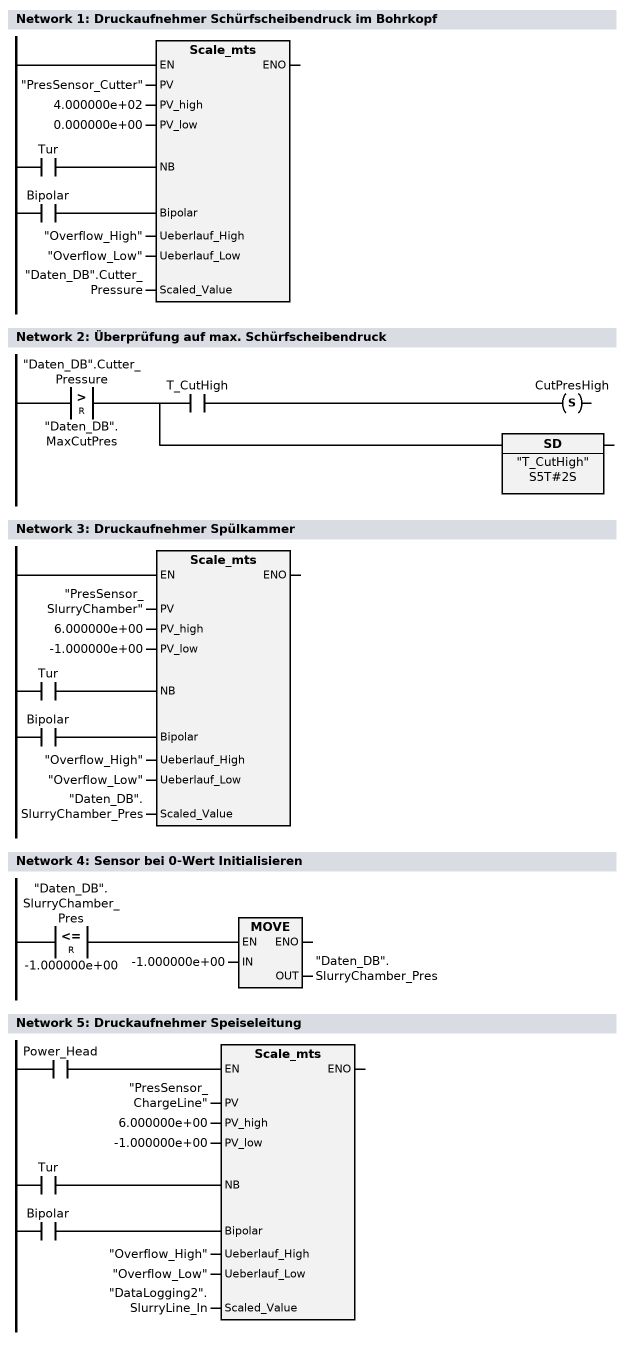
[picture p48: PresSensor_BK networks 1-5]
NETWORK
TITLE = Druckaufnehmer Schürfscheibendruck im Bohrkopf
      A     "Tur";
      =     L 0.0;
      BLD   103;
      A     "Bipolar";
      =     L 0.1;
      BLD   103;
      CALL  "Scale_mts" (
           PV                       := "PresSensor_Cutter",
           PV_high                  := 4.000000e+02,
           PV_low                   := 0.000000e+00,
           NB                       := L 0.0,
           Bipolar                  := L 0.1,
           Ueberlauf_High           := "Overflow_High",
           Ueberlauf_Low            := "Overflow_Low",
           Scaled_Value             := "Daten_DB".Cutter_Pressure);
      NOP   0;
NETWORK
TITLE = Überprüfung auf max. Schürfscheibendruck
      L     "Daten_DB".Cutter_Pressure;
      L     "Daten_DB".MaxCutPres;
      >R;
      =     L 0.0;
      A     L 0.0;
      A     "T_CutHigh";
      S     "CutPresHigh";
      A     L 0.0;
      BLD   102;
      L     S5T#2S;
      SD    "T_CutHigh";
NETWORK
TITLE = Druckaufnehmer Spülkammer
      A     "Tur";
      =     L 0.0;
      BLD   103;
      A     "Bipolar";
      =     L 0.1;
      BLD   103;
      CALL  "Scale_mts" (
           PV                       := "PresSensor_SlurryChamber",
           PV_high                  := 6.000000e+00,
           PV_low                   := -1.000000e+00,
           NB                       := L 0.0,
           Bipolar                  := L 0.1,
           Ueberlauf_High           := "Overflow_High",
           Ueberlauf_Low            := "Overflow_Low",
           Scaled_Value             := "Daten_DB".SlurryChamber_Pres);
      NOP   0;
NETWORK
TITLE = Sensor bei 0-Wert Initialisieren
      A(;
      L     "Daten_DB".SlurryChamber_Pres;
      L     -1.000000e+00;
      <=R;
      );
      JNB   _001;
      L     -1.000000e+00;
      T     "Daten_DB".SlurryChamber_Pres;
_001: NOP   0;
NETWORK
TITLE = Druckaufnehmer Speiseleitung
      A     "Tur";
      =     L 0.0;
      BLD   103;
      A     "Bipolar";
      =     L 0.1;
      BLD   103;
      A     "Power_Head";
      JNB   _002;
      CALL  "Scale_mts" (
           PV                       := "PresSensor_ChargeLine",
           PV_high                  := 6.000000e+00,
           PV_low                   := -1.000000e+00,
           NB                       := L 0.0,
           Bipolar                  := L 0.1,
           Ueberlauf_High           := "Overflow_High",
           Ueberlauf_Low            := "Overflow_Low",
           Scaled_Value             := "DataLogging2".SlurryLine_In);
_002: NOP   0;
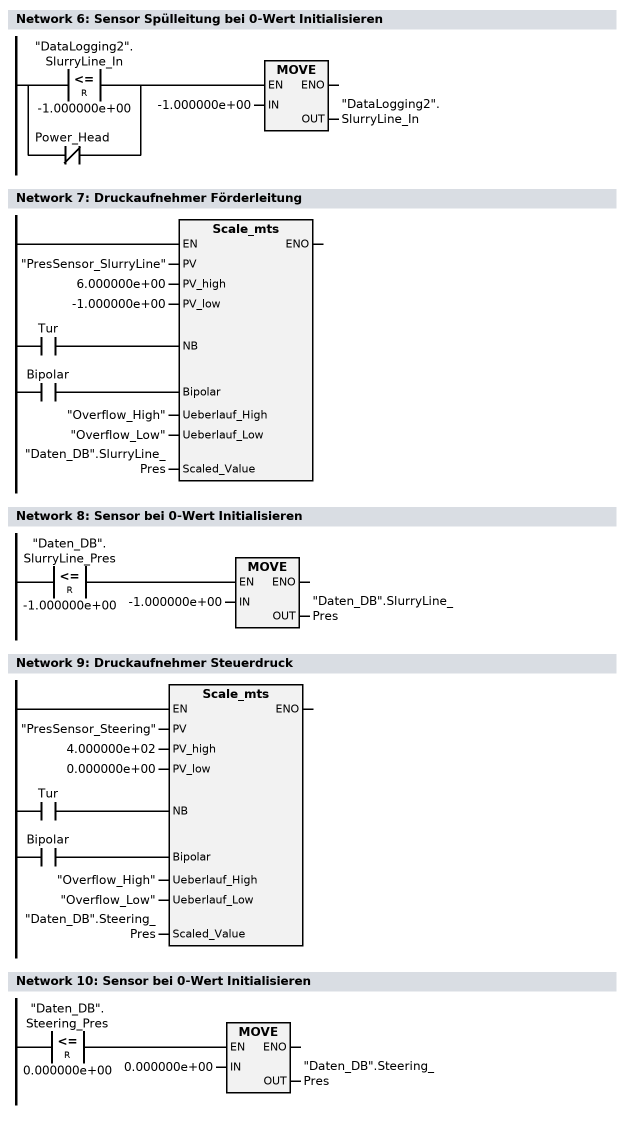
NETWORK
TITLE = Sensor Spülleitung bei 0-Wert Initialisieren
      A(;
      O(;
      L     "DataLogging2".SlurryLine_In;
      L     -1.000000e+00;
      <=R;
      );
      ON    "Power_Head";
      );
      JNB   _003;
      L     -1.000000e+00;
      T     "DataLogging2".SlurryLine_In;
_003: NOP   0;
NETWORK
TITLE = Druckaufnehmer Förderleitung
      A     "Tur";
      =     L 0.0;
      BLD   103;
      A     "Bipolar";
      =     L 0.1;
      BLD   103;
      CALL  "Scale_mts" (
           PV                       := "PresSensor_SlurryLine",
           PV_high                  := 6.000000e+00,
           PV_low                   := -1.000000e+00,
           NB                       := L 0.0,
           Bipolar                  := L 0.1,
           Ueberlauf_High           := "Overflow_High",
           Ueberlauf_Low            := "Overflow_Low",
           Scaled_Value             := "Daten_DB".SlurryLine_Pres);
      NOP   0;
NETWORK
TITLE = Sensor bei 0-Wert Initialisieren
      A(;
      L     "Daten_DB".SlurryLine_Pres;
      L     -1.000000e+00;
      <=R;
      );
      JNB   _004;
      L     -1.000000e+00;
      T     "Daten_DB".SlurryLine_Pres;
_004: NOP   0;
NETWORK
TITLE = Druckaufnehmer Steuerdruck
      A     "Tur";
      =     L 0.0;
      BLD   103;
      A     "Bipolar";
      =     L 0.1;
      BLD   103;
      CALL  "Scale_mts" (
           PV                       := "PresSensor_Steering",
           PV_high                  := 4.000000e+02,
           PV_low                   := 0.000000e+00,
           NB                       := L 0.0,
           Bipolar                  := L 0.1,
           Ueberlauf_High           := "Overflow_High",
           Ueberlauf_Low            := "Overflow_Low",
           Scaled_Value             := "Daten_DB".Steering_Pres);
      NOP   0;
NETWORK
TITLE = Sensor bei 0-Wert Initialisieren
      A(;
      L     "Daten_DB".Steering_Pres;
      L     0.000000e+00;
      <=R;
      );
      JNB   _005;
      L     0.000000e+00;
      T     "Daten_DB".Steering_Pres;
_005: NOP   0;
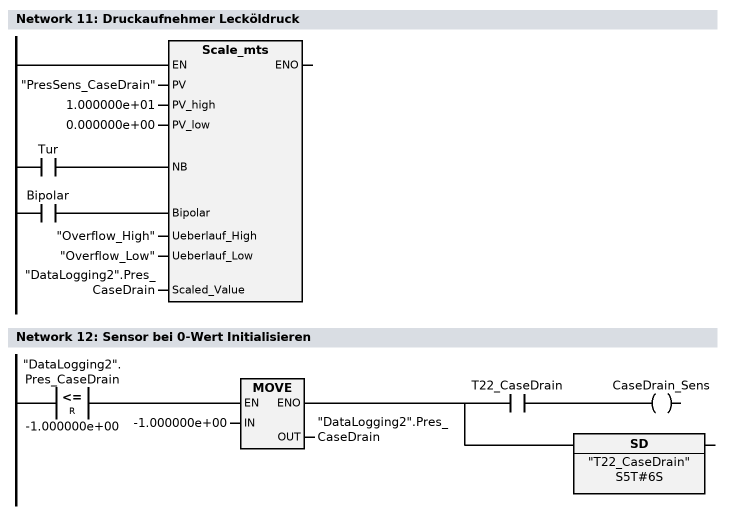
NETWORK
TITLE = Druckaufnehmer Lecköldruck
      A     "Tur";
      =     L 0.0;
      BLD   103;
      A     "Bipolar";
      =     L 0.1;
      BLD   103;
      CALL  "Scale_mts" (
           PV                       := "PresSens_CaseDrain",
           PV_high                  := 1.000000e+01,
           PV_low                   := 0.000000e+00,
           NB                       := L 0.0,
           Bipolar                  := L 0.1,
           Ueberlauf_High           := "Overflow_High",
           Ueberlauf_Low            := "Overflow_Low",
           Scaled_Value             := "DataLogging2".Pres_CaseDrain);
      NOP   0;
NETWORK
TITLE = Sensor bei 0-Wert Initialisieren
      A(;
      L     "DataLogging2".Pres_CaseDrain;
      L     -1.000000e+00;
      <=R;
      );
      JNB   _006;
      L     -1.000000e+00;
      T     "DataLogging2".Pres_CaseDrain;
      SET;
      SAVE;
      CLR;
_006: A     BR;
      =     L 0.0;
      A     L 0.0;
      A     "T22_CaseDrain";
      =     "CaseDrain_Sens";
      A     L 0.0;
      BLD   102;
      L     S5T#6S;
      SD    "T22_CaseDrain";
END_FUNCTION

FUNCTION "Steering cylinder 1" : VOID	// FC 40
TITLE = Funktionen für Steuerzylinder 1
AUTHOR : Simdon
FAMILY : Head
NAME : Cyl_1
VERSION : 0.1
VAR_TEMP
  ist : REAL ;	//Weg ohne Nullabgleich
  Fault : BOOL ;
  Stroke1 : DINT ;
  Stroke : REAL ;
END_VAR
BEGIN
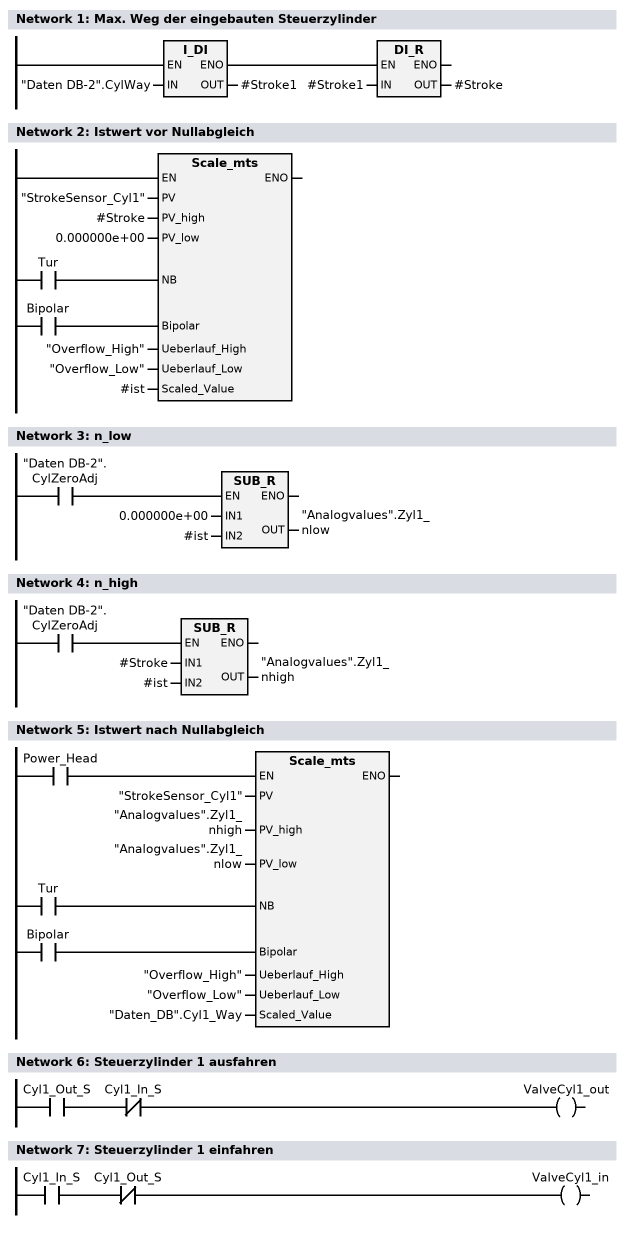
NETWORK
TITLE = Max. Weg der eingebauten Steuerzylinder
      A(;
      L     "Daten DB-2".CylWay;
      ITD;
      T     #Stroke1;
      SET;
      SAVE;
      CLR;
      A     BR;
      );
      JNB   _001;
      L     #Stroke1;
      DTR;
      T     #Stroke;
_001: NOP   0;
NETWORK
TITLE = Istwert vor Nullabgleich
//Istwert des Wegaufnehmers einlesen um die neue Unter- bzw. Obergrenze zur
//Bestimmung des Weges nach dem Nullabgleich. Die Wegaufnehmer liefern ein
//Signal von 4..20 mA.
      A     "Tur";
      =     L 14.0;
      BLD   103;
      A     "Bipolar";
      =     L 14.1;
      BLD   103;
      CALL  "Scale_mts" (
           PV                       := "StrokeSensor_Cyl1",
           PV_high                  := #Stroke,
           PV_low                   := 0.000000e+00,
           NB                       := L 14.0,
           Bipolar                  := L 14.1,
           Ueberlauf_High           := "Overflow_High",
           Ueberlauf_Low            := "Overflow_Low",
           Scaled_Value             := #ist);
      NOP   0;
NETWORK
TITLE = n_low
//Untergrenze der technischen Einheit nach durchgeführtem Nullabgleich.
      A     "Daten DB-2".CylZeroAdj;
      JNB   _002;
      L     0.000000e+00;
      L     #ist;
      -R;
      T     "Analogvalues".Zyl1_nlow;
_002: NOP   0;
NETWORK
TITLE = n_high
//Obergrenze der technischen Einheit nach durchgeführtem Nullabgleich.
      A     "Daten DB-2".CylZeroAdj;
      JNB   _003;
      L     #Stroke;
      L     #ist;
      -R;
      T     "Analogvalues".Zyl1_nhigh;
_003: NOP   0;
NETWORK
TITLE = Istwert nach Nullabgleich
//Istwert des Wegaufnehmers nach durchgeführtem Nullabgleich. Der Rückgabewert 
//liegt
//als Wert mit technischer Einheit (mm) vor.
      A     "Tur";
      =     L 14.0;
      BLD   103;
      A     "Bipolar";
      =     L 14.1;
      BLD   103;
      A     "Power_Head";
      JNB   _004;
      CALL  "Scale_mts" (
           PV                       := "StrokeSensor_Cyl1",
           PV_high                  := "Analogvalues".Zyl1_nhigh,
           PV_low                   := "Analogvalues".Zyl1_nlow,
           NB                       := L 14.0,
           Bipolar                  := L 14.1,
           Ueberlauf_High           := "Overflow_High",
           Ueberlauf_Low            := "Overflow_Low",
           Scaled_Value             := "Daten_DB".Cyl1_Way);
_004: NOP   0;
NETWORK
TITLE = Steuerzylinder 1 ausfahren
      A     "Cyl1_Out_S";
      AN    "Cyl1_In_S";
      =     "ValveCyl1_out";
NETWORK
TITLE = Steuerzylinder 1 einfahren
      A     "Cyl1_In_S";
      AN    "Cyl1_Out_S";
      =     "ValveCyl1_in";
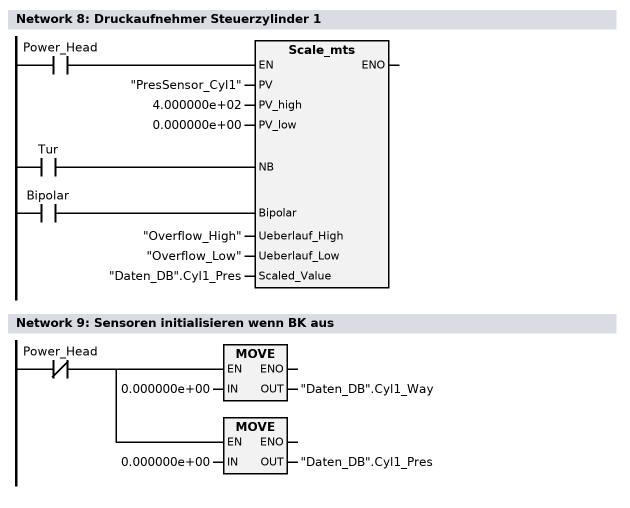
NETWORK
TITLE = Druckaufnehmer Steuerzylinder 1
      A     "Tur";
      =     L 14.0;
      BLD   103;
      A     "Bipolar";
      =     L 14.1;
      BLD   103;
      A     "Power_Head";
      JNB   _005;
      CALL  "Scale_mts" (
           PV                       := "PresSensor_Cyl1",
           PV_high                  := 4.000000e+02,
           PV_low                   := 0.000000e+00,
           NB                       := L 14.0,
           Bipolar                  := L 14.1,
           Ueberlauf_High           := "Overflow_High",
           Ueberlauf_Low            := "Overflow_Low",
           Scaled_Value             := "Daten_DB".Cyl1_Pres);
_005: NOP   0;
NETWORK
TITLE = Sensoren initialisieren wenn BK aus
      AN    "Power_Head";
      =     L 14.0;
      A     L 14.0;
      JNB   _006;
      L     0.000000e+00;
      T     "Daten_DB".Cyl1_Way;
_006: NOP   0;
      A     L 14.0;
      JNB   _007;
      L     0.000000e+00;
      T     "Daten_DB".Cyl1_Pres;
_007: NOP   0;
END_FUNCTION

FUNCTION "Steering cylinder 2" : VOID	// FC 41
TITLE = Funktionen für Steuerzylinder 2
AUTHOR : Simdon
FAMILY : Head
NAME : Cyl_2
VERSION : 0.1
VAR_TEMP
  ist : REAL ;	//Weg ohne Nullabgleich
  Fault : BOOL ;
  Stroke1 : DINT ;
  Stroke : REAL ;
END_VAR
BEGIN
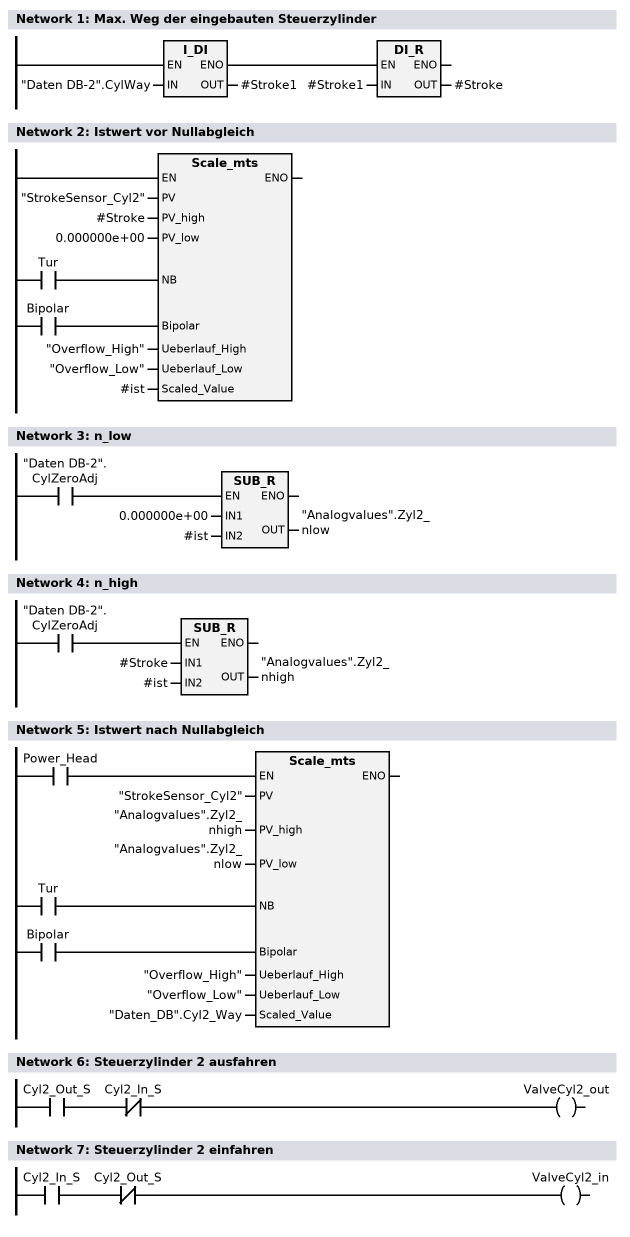
NETWORK
TITLE = Max. Weg der eingebauten Steuerzylinder
      A(;
      L     "Daten DB-2".CylWay;
      ITD;
      T     #Stroke1;
      SET;
      SAVE;
      CLR;
      A     BR;
      );
      JNB   _001;
      L     #Stroke1;
      DTR;
      T     #Stroke;
_001: NOP   0;
NETWORK
TITLE = Istwert vor Nullabgleich
//Istwert des Wegaufnehmers einlesen um die neue Unter- bzw. Obergrenze zur
//Bestimmung des Weges nach dem Nullabgleich. Die Wegaufnehmer liefern ein
//Signal von 4..20 mA.
      A     "Tur";
      =     L 14.0;
      BLD   103;
      A     "Bipolar";
      =     L 14.1;
      BLD   103;
      CALL  "Scale_mts" (
           PV                       := "StrokeSensor_Cyl2",
           PV_high                  := #Stroke,
           PV_low                   := 0.000000e+00,
           NB                       := L 14.0,
           Bipolar                  := L 14.1,
           Ueberlauf_High           := "Overflow_High",
           Ueberlauf_Low            := "Overflow_Low",
           Scaled_Value             := #ist);
      NOP   0;
NETWORK
TITLE = n_low
//Untergrenze der technischen Einheit nach durchgeführtem Nullabgleich.
      A     "Daten DB-2".CylZeroAdj;
      JNB   _002;
      L     0.000000e+00;
      L     #ist;
      -R;
      T     "Analogvalues".Zyl2_nlow;
_002: NOP   0;
NETWORK
TITLE = n_high
//Obergrenze der technischen Einheit nach durchgeführtem Nullabgleich.
      A     "Daten DB-2".CylZeroAdj;
      JNB   _003;
      L     #Stroke;
      L     #ist;
      -R;
      T     "Analogvalues".Zyl2_nhigh;
_003: NOP   0;
NETWORK
TITLE = Istwert nach Nullabgleich
//Istwert des Wegaufnehmers nach durchgeführtem Nullabgleich. Der Rückgabewert 
//liegt
//als Wert mit technischer Einheit (mm) vor.
      A     "Tur";
      =     L 14.0;
      BLD   103;
      A     "Bipolar";
      =     L 14.1;
      BLD   103;
      A     "Power_Head";
      JNB   _004;
      CALL  "Scale_mts" (
           PV                       := "StrokeSensor_Cyl2",
           PV_high                  := "Analogvalues".Zyl2_nhigh,
           PV_low                   := "Analogvalues".Zyl2_nlow,
           NB                       := L 14.0,
           Bipolar                  := L 14.1,
           Ueberlauf_High           := "Overflow_High",
           Ueberlauf_Low            := "Overflow_Low",
           Scaled_Value             := "Daten_DB".Cyl2_Way);
_004: NOP   0;
NETWORK
TITLE = Steuerzylinder 2 ausfahren
      A     "Cyl2_Out_S";
      AN    "Cyl2_In_S";
      =     "ValveCyl2_out";
NETWORK
TITLE = Steuerzylinder 2 einfahren
      A     "Cyl2_In_S";
      AN    "Cyl2_Out_S";
      =     "ValveCyl2_in";
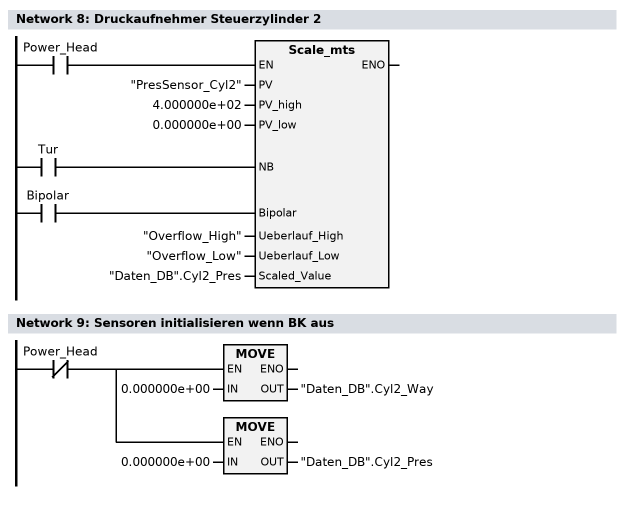
NETWORK
TITLE = Druckaufnehmer Steuerzylinder 2
      A     "Tur";
      =     L 14.0;
      BLD   103;
      A     "Bipolar";
      =     L 14.1;
      BLD   103;
      A     "Power_Head";
      JNB   _005;
      CALL  "Scale_mts" (
           PV                       := "PresSensor_Cyl2",
           PV_high                  := 4.000000e+02,
           PV_low                   := 0.000000e+00,
           NB                       := L 14.0,
           Bipolar                  := L 14.1,
           Ueberlauf_High           := "Overflow_High",
           Ueberlauf_Low            := "Overflow_Low",
           Scaled_Value             := "Daten_DB".Cyl2_Pres);
_005: NOP   0;
NETWORK
TITLE = Sensoren initialisieren wenn BK aus
      AN    "Power_Head";
      =     L 14.0;
      A     L 14.0;
      JNB   _006;
      L     0.000000e+00;
      T     "Daten_DB".Cyl2_Way;
_006: NOP   0;
      A     L 14.0;
      JNB   _007;
      L     0.000000e+00;
      T     "Daten_DB".Cyl2_Pres;
_007: NOP   0;
END_FUNCTION

FUNCTION "Steering cylinder 3" : VOID	// FC 42
TITLE = Funktionen für Steuerzylinder 3
AUTHOR : Simdon
FAMILY : Head
NAME : Cyl_3
VERSION : 0.1
VAR_TEMP
  ist : REAL ;	//Weg ohne Nullabgleich
  Fault : BOOL ;
  eins : INT ;
  Stroke1 : DINT ;
  Stroke : REAL ;
END_VAR
BEGIN
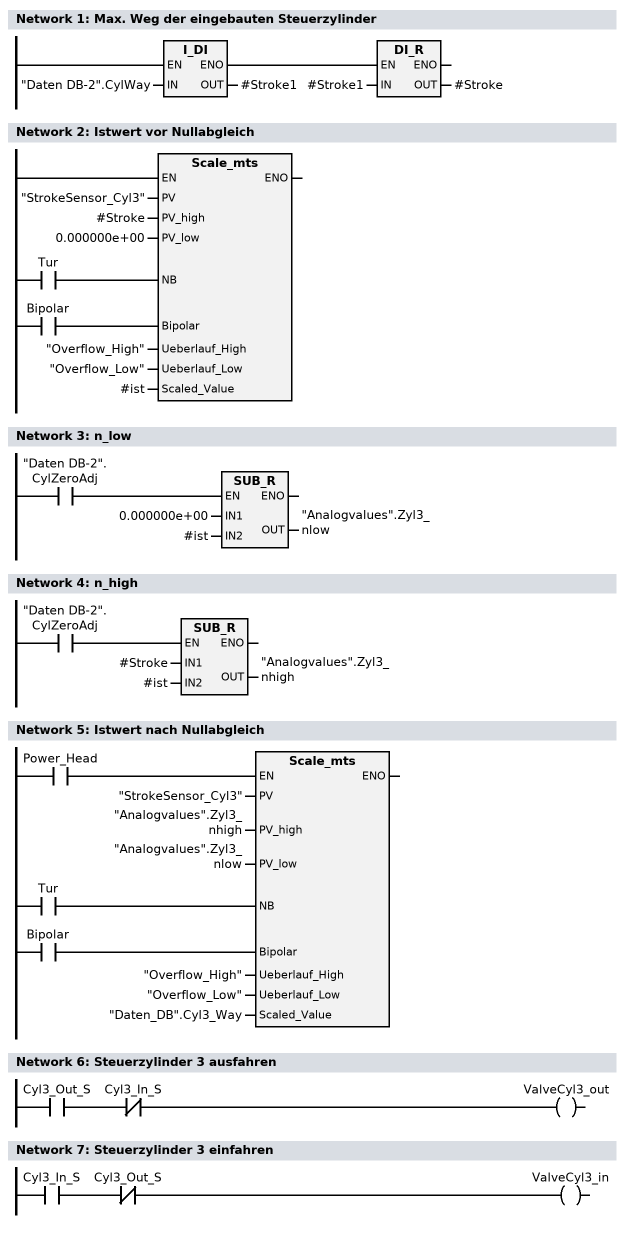
NETWORK
TITLE = Max. Weg der eingebauten Steuerzylinder
      A(;
      L     "Daten DB-2".CylWay;
      ITD;
      T     #Stroke1;
      SET;
      SAVE;
      CLR;
      A     BR;
      );
      JNB   _001;
      L     #Stroke1;
      DTR;
      T     #Stroke;
_001: NOP   0;
NETWORK
TITLE = Istwert vor Nullabgleich
//Istwert des Wegaufnehmers einlesen um die neue Unter- bzw. Obergrenze zur
//Bestimmung des Weges nach dem Nullabgleich. Die Wegaufnehmer liefern ein
//Signal von 4..20 mA.
      A     "Tur";
      =     L 16.0;
      BLD   103;
      A     "Bipolar";
      =     L 16.1;
      BLD   103;
      CALL  "Scale_mts" (
           PV                       := "StrokeSensor_Cyl3",
           PV_high                  := #Stroke,
           PV_low                   := 0.000000e+00,
           NB                       := L 16.0,
           Bipolar                  := L 16.1,
           Ueberlauf_High           := "Overflow_High",
           Ueberlauf_Low            := "Overflow_Low",
           Scaled_Value             := #ist);
      NOP   0;
NETWORK
TITLE = n_low
//Untergrenze der technischen Einheit nach durchgeführtem Nullabgleich.
      A     "Daten DB-2".CylZeroAdj;
      JNB   _002;
      L     0.000000e+00;
      L     #ist;
      -R;
      T     "Analogvalues".Zyl3_nlow;
_002: NOP   0;
NETWORK
TITLE = n_high
//Obergrenze der technischen Einheit nach durchgeführtem Nullabgleich.
      A     "Daten DB-2".CylZeroAdj;
      JNB   _003;
      L     #Stroke;
      L     #ist;
      -R;
      T     "Analogvalues".Zyl3_nhigh;
_003: NOP   0;
NETWORK
TITLE = Istwert nach Nullabgleich
//Istwert des Wegaufnehmers nach durchgeführtem Nullabgleich. Der Rückgabewert 
//liegt
//als Wert mit technischer Einheit (mm) vor.
      A     "Tur";
      =     L 16.0;
      BLD   103;
      A     "Bipolar";
      =     L 16.1;
      BLD   103;
      A     "Power_Head";
      JNB   _004;
      CALL  "Scale_mts" (
           PV                       := "StrokeSensor_Cyl3",
           PV_high                  := "Analogvalues".Zyl3_nhigh,
           PV_low                   := "Analogvalues".Zyl3_nlow,
           NB                       := L 16.0,
           Bipolar                  := L 16.1,
           Ueberlauf_High           := "Overflow_High",
           Ueberlauf_Low            := "Overflow_Low",
           Scaled_Value             := "Daten_DB".Cyl3_Way);
_004: NOP   0;
NETWORK
TITLE = Steuerzylinder 3 ausfahren
      A     "Cyl3_Out_S";
      AN    "Cyl3_In_S";
      =     "ValveCyl3_out";
NETWORK
TITLE = Steuerzylinder 3 einfahren
      A     "Cyl3_In_S";
      AN    "Cyl3_Out_S";
      =     "ValveCyl3_in";
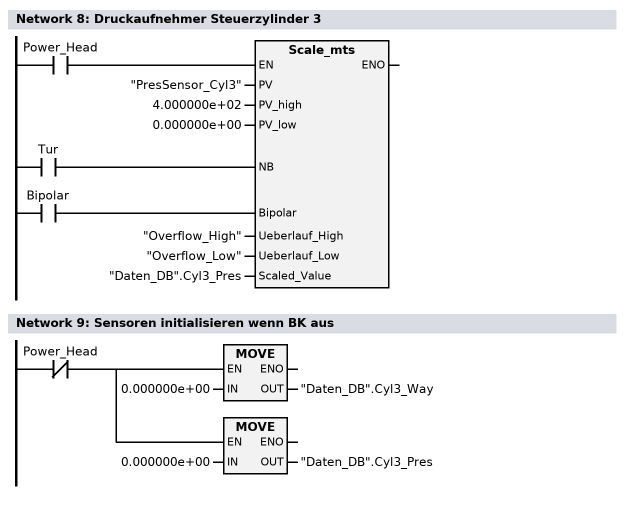
NETWORK
TITLE = Druckaufnehmer Steuerzylinder 3
      A     "Tur";
      =     L 16.0;
      BLD   103;
      A     "Bipolar";
      =     L 16.1;
      BLD   103;
      A     "Power_Head";
      JNB   _005;
      CALL  "Scale_mts" (
           PV                       := "PresSensor_Cyl3",
           PV_high                  := 4.000000e+02,
           PV_low                   := 0.000000e+00,
           NB                       := L 16.0,
           Bipolar                  := L 16.1,
           Ueberlauf_High           := "Overflow_High",
           Ueberlauf_Low            := "Overflow_Low",
           Scaled_Value             := "Daten_DB".Cyl3_Pres);
_005: NOP   0;
NETWORK
TITLE = Sensoren initialisieren wenn BK aus
      AN    "Power_Head";
      =     L 16.0;
      A     L 16.0;
      JNB   _006;
      L     0.000000e+00;
      T     "Daten_DB".Cyl3_Way;
_006: NOP   0;
      A     L 16.0;
      JNB   _007;
      L     0.000000e+00;
      T     "Daten_DB".Cyl3_Pres;
_007: NOP   0;
END_FUNCTION

FUNCTION "Wing" : VOID	// FC 43
TITLE = Funktionen für Flossenzylinder
AUTHOR : Simdon
FAMILY : Head
NAME : Wing
VERSION : 0.1
VAR_TEMP
  ist : REAL ;	//Weg ohne Nullabgleich
  Fault : BOOL ;
END_VAR
BEGIN
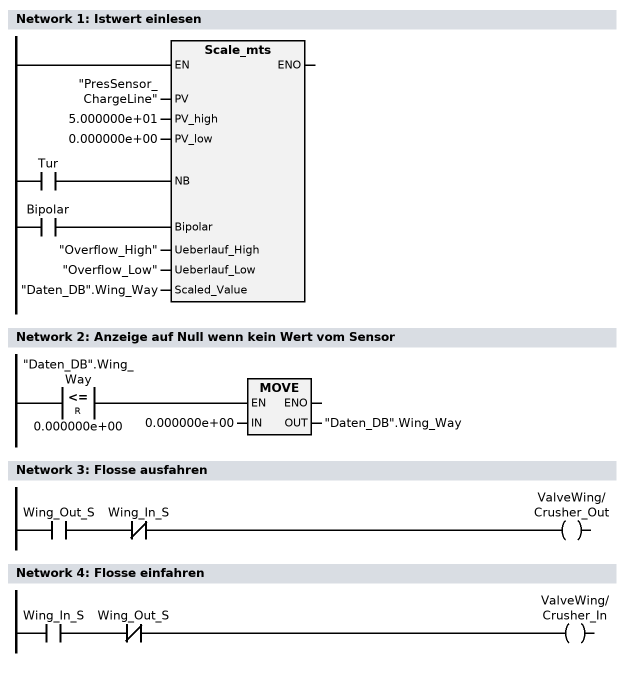
NETWORK
TITLE = Istwert einlesen
//Istwert des Wegaufnehmers nach durchgeführtem Nullabgleich. Der Rückgabewert 
//liegt
//als Wert mit technischer Einheit (mm) vor.
      A     "Tur";
      =     L 5.0;
      BLD   103;
      A     "Bipolar";
      =     L 5.1;
      BLD   103;
      CALL  "Scale_mts" (
           PV                       := "PresSensor_ChargeLine",
           PV_high                  := 5.000000e+01,
           PV_low                   := 0.000000e+00,
           NB                       := L 5.0,
           Bipolar                  := L 5.1,
           Ueberlauf_High           := "Overflow_High",
           Ueberlauf_Low            := "Overflow_Low",
           Scaled_Value             := "Daten_DB".Wing_Way);
      NOP   0;
NETWORK
TITLE = Anzeige auf Null wenn kein Wert vom Sensor
      A(;
      L     "Daten_DB".Wing_Way;
      L     0.000000e+00;
      <=R;
      );
      JNB   _001;
      L     0.000000e+00;
      T     "Daten_DB".Wing_Way;
_001: NOP   0;
NETWORK
TITLE = Flosse ausfahren
      A     "Wing_Out_S";
      AN    "Wing_In_S";
      =     "ValveWing/Crusher_Out";
NETWORK
TITLE = Flosse einfahren
      A     "Wing_In_S";
      AN    "Wing_Out_S";
      =     "ValveWing/Crusher_In";
END_FUNCTION

FUNCTION "Locking cylinder" : VOID	// FC 44
TITLE = Verbindungszylinder für Bohrkopf und Nachläufer
AUTHOR : Simdon
FAMILY : Head
NAME : VerbCyl
VERSION : 0.1
BEGIN
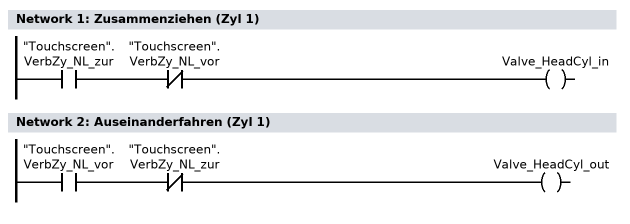
NETWORK
TITLE = Zusammenziehen (Zyl 1)
      A     "Touchscreen".VerbZy_NL_zur;
      AN    "Touchscreen".VerbZy_NL_vor;
      =     "Valve_HeadCyl_in";
NETWORK
TITLE = Auseinanderfahren (Zyl 1)
      A     "Touchscreen".VerbZy_NL_vor;
      AN    "Touchscreen".VerbZy_NL_zur;
      =     "Valve_HeadCyl_out";
END_FUNCTION

FUNCTION "Flowmeter" : VOID	// FC 50
TITLE = Durchflußmengenmessung in der Spülleitung
AUTHOR : Simdon
FAMILY : Slurry
NAME : Flow
VERSION : 0.1
VAR_TEMP
  Max_Flow : REAL ;
END_VAR
BEGIN
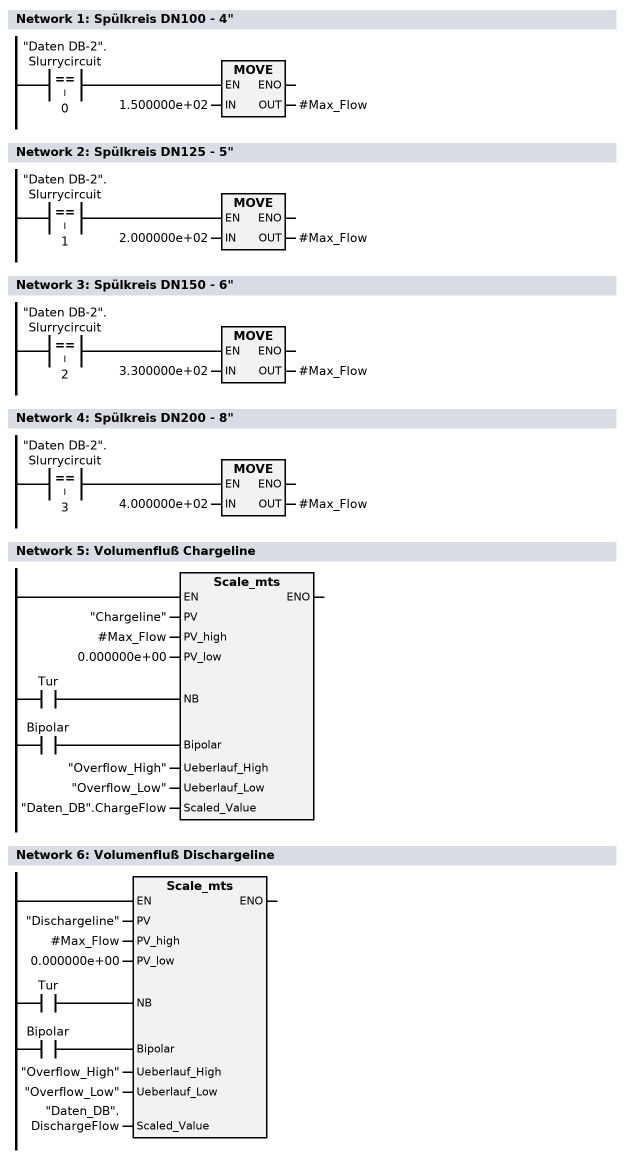
NETWORK
TITLE = Spülkreis DN100 - 4"
      A(;
      L     "Daten DB-2".Slurrycircuit;
      L     0;
      ==I;
      );
      JNB   _001;
      L     1.500000e+02;
      T     #Max_Flow;
_001: NOP   0;
NETWORK
TITLE = Spülkreis DN125 - 5"
      A(;
      L     "Daten DB-2".Slurrycircuit;
      L     1;
      ==I;
      );
      JNB   _002;
      L     2.000000e+02;
      T     #Max_Flow;
_002: NOP   0;
NETWORK
TITLE = Spülkreis DN150 - 6"
      A(;
      L     "Daten DB-2".Slurrycircuit;
      L     2;
      ==I;
      );
      JNB   _003;
      L     3.300000e+02;
      T     #Max_Flow;
_003: NOP   0;
NETWORK
TITLE = Spülkreis DN200 - 8"
      A(;
      L     "Daten DB-2".Slurrycircuit;
      L     3;
      ==I;
      );
      JNB   _004;
      L     4.000000e+02;
      T     #Max_Flow;
_004: NOP   0;
NETWORK
TITLE = Volumenfluß Chargeline
      A     "Tur";
      =     L 4.0;
      BLD   103;
      A     "Bipolar";
      =     L 4.1;
      BLD   103;
      CALL  "Scale_mts" (
           PV                       := "Chargeline",
           PV_high                  := #Max_Flow,
           PV_low                   := 0.000000e+00,
           NB                       := L 4.0,
           Bipolar                  := L 4.1,
           Ueberlauf_High           := "Overflow_High",
           Ueberlauf_Low            := "Overflow_Low",
           Scaled_Value             := "Daten_DB".ChargeFlow);
      NOP   0;
NETWORK
TITLE = Volumenfluß Dischargeline
      A     "Tur";
      =     L 4.0;
      BLD   103;
      A     "Bipolar";
      =     L 4.1;
      BLD   103;
      CALL  "Scale_mts" (
           PV                       := "Dischargeline",
           PV_high                  := #Max_Flow,
           PV_low                   := 0.000000e+00,
           NB                       := L 4.0,
           Bipolar                  := L 4.1,
           Ueberlauf_High           := "Overflow_High",
           Ueberlauf_Low            := "Overflow_Low",
           Scaled_Value             := "Daten_DB".DischargeFlow);
      NOP   0;
END_FUNCTION

FUNCTION "Jet -Bypass" : VOID	// FC 51
TITLE = Steuerung Jet und Bypass
AUTHOR : Simdon
FAMILY : Head
NAME : Jet_Byp
VERSION : 1.0
BEGIN
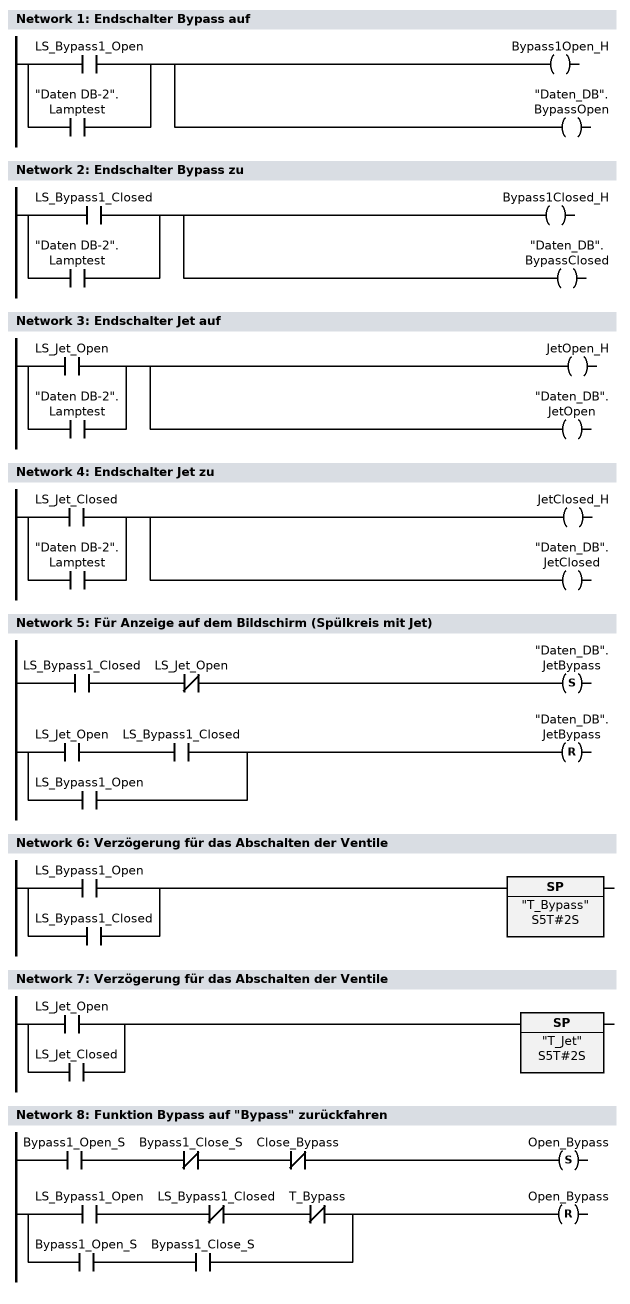
NETWORK
TITLE = Endschalter Bypass auf
      O     "LS_Bypass1_Open";
      O     "Daten DB-2".Lamptest;
      =     "Bypass1Open_H";
      =     "Daten_DB".BypassOpen;
NETWORK
TITLE = Endschalter Bypass zu
      O     "LS_Bypass1_Closed";
      O     "Daten DB-2".Lamptest;
      =     "Bypass1Closed_H";
      =     "Daten_DB".BypassClosed;
NETWORK
TITLE = Endschalter Jet auf
      O     "LS_Jet_Open";
      O     "Daten DB-2".Lamptest;
      =     "JetOpen_H";
      =     "Daten_DB".JetOpen;
NETWORK
TITLE = Endschalter Jet zu
      O     "LS_Jet_Closed";
      O     "Daten DB-2".Lamptest;
      =     "JetClosed_H";
      =     "Daten_DB".JetClosed;
NETWORK
TITLE = Für Anzeige auf dem Bildschirm (Spülkreis mit Jet)
      A     "LS_Bypass1_Closed";
      AN    "LS_Jet_Open";
      S     "Daten_DB".JetBypass;
      A(;
      A     "LS_Jet_Open";
      A     "LS_Bypass1_Closed";
      O     "LS_Bypass1_Open";
      );
      R     "Daten_DB".JetBypass;
      NOP   0;
NETWORK
TITLE = Verzögerung für das Abschalten der Ventile
      O     "LS_Bypass1_Open";
      O     "LS_Bypass1_Closed";
      L     S5T#2S;
      SP    "T_Bypass";
NETWORK
TITLE = Verzögerung für das Abschalten der Ventile
      O     "LS_Jet_Open";
      O     "LS_Jet_Closed";
      L     S5T#2S;
      SP    "T_Jet";
NETWORK
TITLE = Funktion Bypass auf "Bypass" zurückfahren
      A     "Bypass1_Open_S";
      AN    "Bypass1_Close_S";
      AN    "Close_Bypass";
      S     "Open_Bypass";
      A(;
      A     "LS_Bypass1_Open";
      AN    "LS_Bypass1_Closed";
      AN    "T_Bypass";
      O;
      A     "Bypass1_Open_S";
      A     "Bypass1_Close_S";
      );
      R     "Open_Bypass";
      NOP   0;
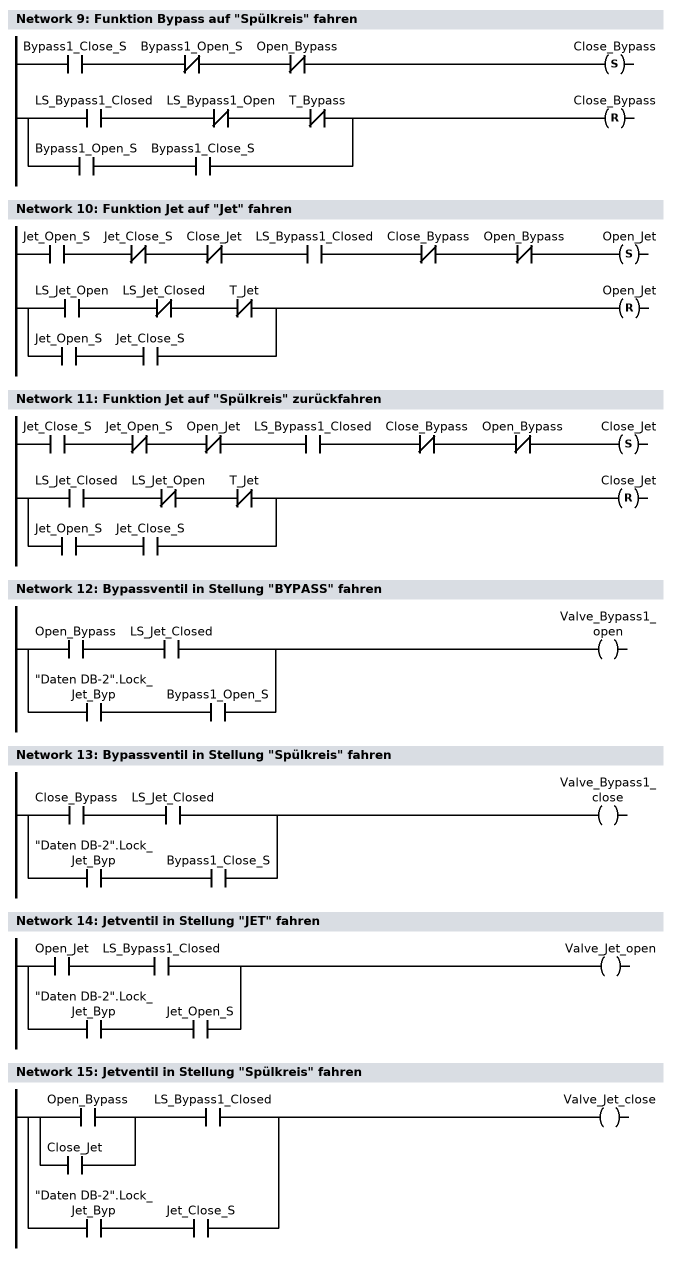
NETWORK
TITLE = Funktion Bypass auf "Spülkreis" fahren
      A     "Bypass1_Close_S";
      AN    "Bypass1_Open_S";
      AN    "Open_Bypass";
      S     "Close_Bypass";
      A(;
      A     "LS_Bypass1_Closed";
      AN    "LS_Bypass1_Open";
      AN    "T_Bypass";
      O;
      A     "Bypass1_Open_S";
      A     "Bypass1_Close_S";
      );
      R     "Close_Bypass";
      NOP   0;
NETWORK
TITLE = Funktion Jet auf "Jet" fahren
      A     "Jet_Open_S";
      AN    "Jet_Close_S";
      AN    "Close_Jet";
      A     "LS_Bypass1_Closed";
      AN    "Close_Bypass";
      AN    "Open_Bypass";
      S     "Open_Jet";
      A(;
      A     "LS_Jet_Open";
      AN    "LS_Jet_Closed";
      AN    "T_Jet";
      O;
      A     "Jet_Open_S";
      A     "Jet_Close_S";
      );
      R     "Open_Jet";
      NOP   0;
NETWORK
TITLE = Funktion Jet auf "Spülkreis" zurückfahren
      A     "Jet_Close_S";
      AN    "Jet_Open_S";
      AN    "Open_Jet";
      A     "LS_Bypass1_Closed";
      AN    "Close_Bypass";
      AN    "Open_Bypass";
      S     "Close_Jet";
      A(;
      A     "LS_Jet_Closed";
      AN    "LS_Jet_Open";
      AN    "T_Jet";
      O;
      A     "Jet_Open_S";
      A     "Jet_Close_S";
      );
      R     "Close_Jet";
      NOP   0;
NETWORK
TITLE = Bypassventil in Stellung "BYPASS" fahren
      A     "Open_Bypass";
      A     "LS_Jet_Closed";
      O;
      A     "Daten DB-2".Lock_Jet_Byp;
      A     "Bypass1_Open_S";
      =     "Valve_Bypass1_open";
NETWORK
TITLE = Bypassventil in Stellung "Spülkreis" fahren
      A     "Close_Bypass";
      A     "LS_Jet_Closed";
      O;
      A     "Daten DB-2".Lock_Jet_Byp;
      A     "Bypass1_Close_S";
      =     "Valve_Bypass1_close";
NETWORK
TITLE = Jetventil in Stellung "JET" fahren
      A     "Open_Jet";
      A     "LS_Bypass1_Closed";
      O;
      A     "Daten DB-2".Lock_Jet_Byp;
      A     "Jet_Open_S";
      =     "Valve_Jet_open";
NETWORK
TITLE = Jetventil in Stellung "Spülkreis" fahren
      A(;
      O     "Open_Bypass";
      O     "Close_Jet";
      );
      A     "LS_Bypass1_Closed";
      O;
      A     "Daten DB-2".Lock_Jet_Byp;
      A     "Jet_Close_S";
      =     "Valve_Jet_close";
END_FUNCTION

FUNCTION "Interjack1" : VOID	// FC 55
TITLE = Steuerung Dehner #1
AUTHOR : Simdon
FAMILY : Presse
NAME : Inter1
VERSION : 0.1
VAR_TEMP
  Inter_Release : BOOL ;
  Inter1_okay : BOOL ;
  Druck_Inter1 : REAL ;
END_VAR
BEGIN
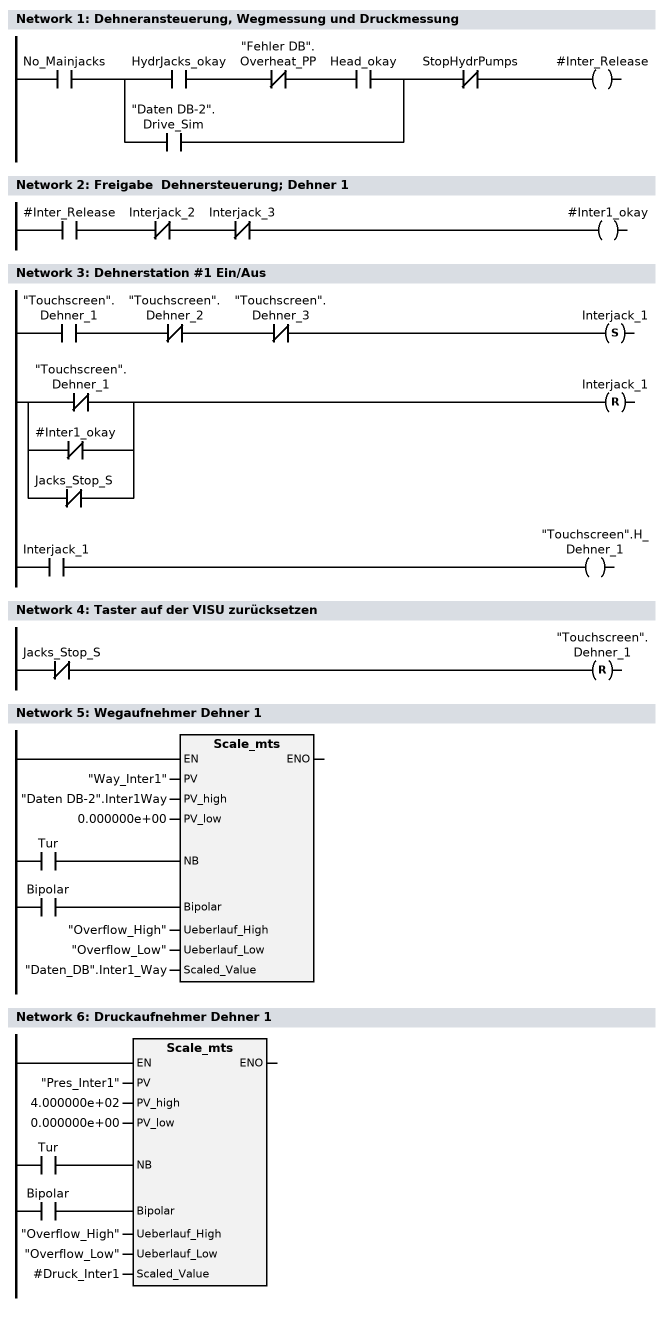
NETWORK
TITLE = Dehneransteuerung, Wegmessung und Druckmessung
      A     "No_Mainjacks";
      A(;
      A     "HydrJacks_okay";
      AN    "Fehler DB".Overheat_PP;
      A     "Head_okay";
      O     "Daten DB-2".Drive_Sim;
      );
      AN    "StopHydrPumps";
      =     #Inter_Release;
NETWORK
TITLE = Freigabe  Dehnersteuerung; Dehner 1
      A     #Inter_Release;
      AN    "Interjack_2";
      AN    "Interjack_3";
      =     #Inter1_okay;
NETWORK
TITLE = Dehnerstation #1 Ein/Aus
      A     "Touchscreen".Dehner_1;
      AN    "Touchscreen".Dehner_2;
      AN    "Touchscreen".Dehner_3;
      S     "Interjack_1";
      A(;
      ON    "Touchscreen".Dehner_1;
      ON    #Inter1_okay;
      ON    "Jacks_Stop_S";
      );
      R     "Interjack_1";
      A     "Interjack_1";
      =     "Touchscreen".H_Dehner_1;
NETWORK
TITLE = Taster auf der VISU zurücksetzen
      AN    "Jacks_Stop_S";
      R     "Touchscreen".Dehner_1;
NETWORK
TITLE = Wegaufnehmer Dehner 1
      A     "Tur";
      =     L 6.0;
      BLD   103;
      A     "Bipolar";
      =     L 6.1;
      BLD   103;
      CALL  "Scale_mts" (
           PV                       := "Way_Inter1",
           PV_high                  := "Daten DB-2".Inter1Way,
           PV_low                   := 0.000000e+00,
           NB                       := L 6.0,
           Bipolar                  := L 6.1,
           Ueberlauf_High           := "Overflow_High",
           Ueberlauf_Low            := "Overflow_Low",
           Scaled_Value             := "Daten_DB".Inter1_Way);
      NOP   0;
NETWORK
TITLE = Druckaufnehmer Dehner 1
      A     "Tur";
      =     L 6.0;
      BLD   103;
      A     "Bipolar";
      =     L 6.1;
      BLD   103;
      CALL  "Scale_mts" (
           PV                       := "Pres_Inter1",
           PV_high                  := 4.000000e+02,
           PV_low                   := 0.000000e+00,
           NB                       := L 6.0,
           Bipolar                  := L 6.1,
           Ueberlauf_High           := "Overflow_High",
           Ueberlauf_Low            := "Overflow_Low",
           Scaled_Value             := #Druck_Inter1);
      NOP   0;
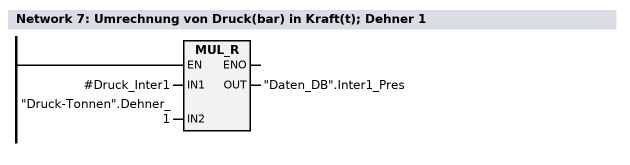
NETWORK
TITLE = Umrechnung von Druck(bar) in Kraft(t); Dehner 1
      L     #Druck_Inter1;
      L     "Druck-Tonnen".Dehner_1;
      *R;
      T     "Daten_DB".Inter1_Pres;
      NOP   0;
END_FUNCTION

FUNCTION "Interjack2" : VOID	// FC 56
TITLE = Steuerung Dehner 2
AUTHOR : Simdon
FAMILY : Presse
NAME : Inter2
VERSION : 0.1
VAR_TEMP
  Inter_Release : BOOL ;	//Freigabe Dehnersteuerung
  Inter2_okay : BOOL ;	//Freigabe Dehner 2
  Druck_Inter2 : REAL ;	//Druck Dehnerstation 2
END_VAR
BEGIN
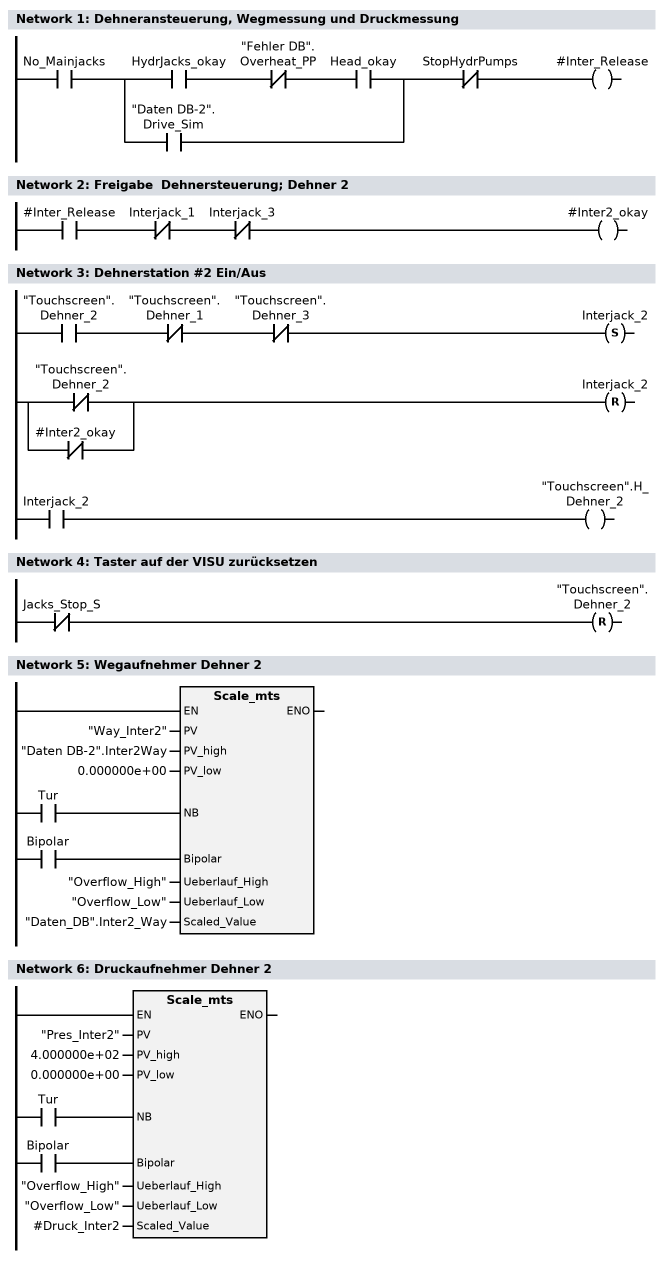
NETWORK
TITLE = Dehneransteuerung, Wegmessung und Druckmessung
      A     "No_Mainjacks";
      A(;
      A     "HydrJacks_okay";
      AN    "Fehler DB".Overheat_PP;
      A     "Head_okay";
      O     "Daten DB-2".Drive_Sim;
      );
      AN    "StopHydrPumps";
      =     #Inter_Release;
NETWORK
TITLE = Freigabe  Dehnersteuerung; Dehner 2
      A     #Inter_Release;
      AN    "Interjack_1";
      AN    "Interjack_3";
      =     #Inter2_okay;
NETWORK
TITLE = Dehnerstation #2 Ein/Aus
      A     "Touchscreen".Dehner_2;
      AN    "Touchscreen".Dehner_1;
      AN    "Touchscreen".Dehner_3;
      S     "Interjack_2";
      A(;
      ON    "Touchscreen".Dehner_2;
      ON    #Inter2_okay;
      );
      R     "Interjack_2";
      A     "Interjack_2";
      =     "Touchscreen".H_Dehner_2;
NETWORK
TITLE = Taster auf der VISU zurücksetzen
      AN    "Jacks_Stop_S";
      R     "Touchscreen".Dehner_2;
NETWORK
TITLE = Wegaufnehmer Dehner 2
      A     "Tur";
      =     L 6.0;
      BLD   103;
      A     "Bipolar";
      =     L 6.1;
      BLD   103;
      CALL  "Scale_mts" (
           PV                       := "Way_Inter2",
           PV_high                  := "Daten DB-2".Inter2Way,
           PV_low                   := 0.000000e+00,
           NB                       := L 6.0,
           Bipolar                  := L 6.1,
           Ueberlauf_High           := "Overflow_High",
           Ueberlauf_Low            := "Overflow_Low",
           Scaled_Value             := "Daten_DB".Inter2_Way);
      NOP   0;
NETWORK
TITLE = Druckaufnehmer Dehner 2
      A     "Tur";
      =     L 6.0;
      BLD   103;
      A     "Bipolar";
      =     L 6.1;
      BLD   103;
      CALL  "Scale_mts" (
           PV                       := "Pres_Inter2",
           PV_high                  := 4.000000e+02,
           PV_low                   := 0.000000e+00,
           NB                       := L 6.0,
           Bipolar                  := L 6.1,
           Ueberlauf_High           := "Overflow_High",
           Ueberlauf_Low            := "Overflow_Low",
           Scaled_Value             := #Druck_Inter2);
      NOP   0;
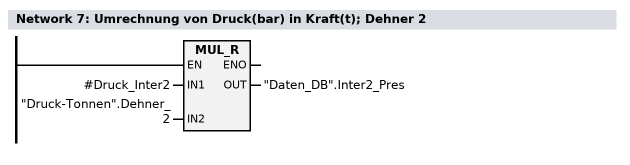
NETWORK
TITLE = Umrechnung von Druck(bar) in Kraft(t); Dehner 2
      L     #Druck_Inter2;
      L     "Druck-Tonnen".Dehner_2;
      *R;
      T     "Daten_DB".Inter2_Pres;
      NOP   0;
END_FUNCTION

FUNCTION "Interjack3" : VOID	// FC 57
TITLE = Steuerung Dehner 3
AUTHOR : Simdon
FAMILY : Presse
NAME : Inter3
VERSION : 0.1
VAR_TEMP
  Inter_Release : BOOL ;	//Freigabe Dehnersteuerung
  Inter3_okay : BOOL ;
  Druck_Inter3 : REAL ;
END_VAR
BEGIN
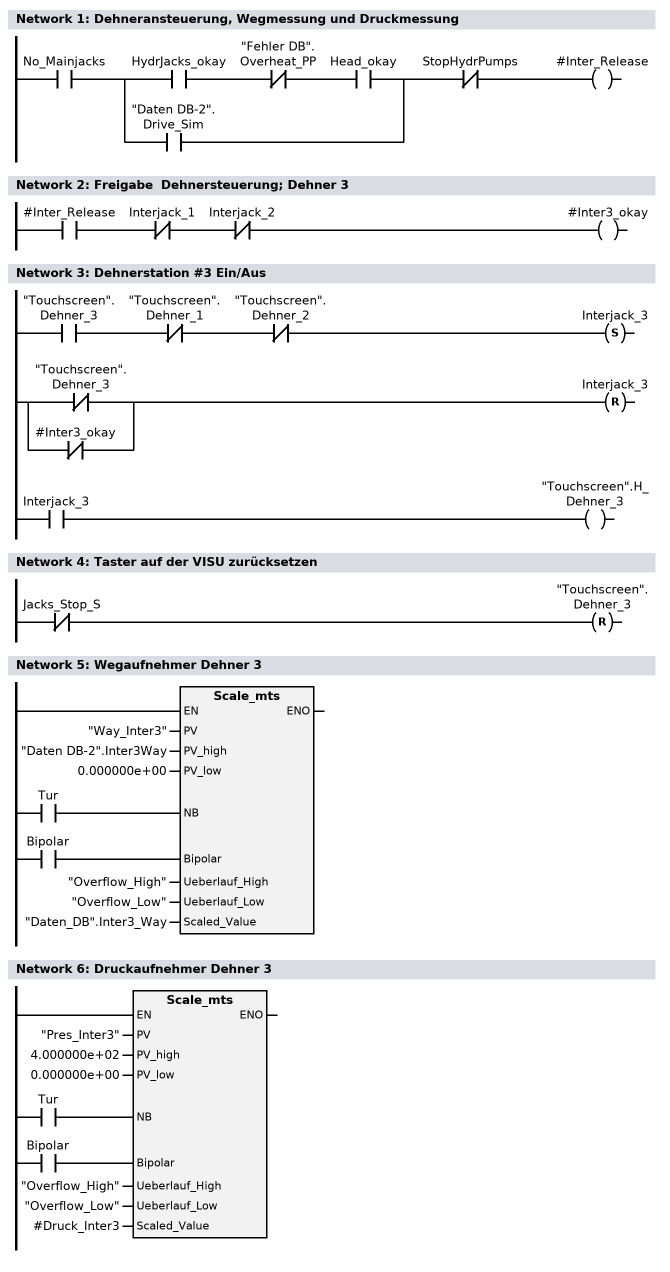
NETWORK
TITLE = Dehneransteuerung, Wegmessung und Druckmessung
      A     "No_Mainjacks";
      A(;
      A     "HydrJacks_okay";
      AN    "Fehler DB".Overheat_PP;
      A     "Head_okay";
      O     "Daten DB-2".Drive_Sim;
      );
      AN    "StopHydrPumps";
      =     #Inter_Release;
NETWORK
TITLE = Freigabe  Dehnersteuerung; Dehner 3
      A     #Inter_Release;
      AN    "Interjack_1";
      AN    "Interjack_2";
      =     #Inter3_okay;
NETWORK
TITLE = Dehnerstation #3 Ein/Aus
      A     "Touchscreen".Dehner_3;
      AN    "Touchscreen".Dehner_1;
      AN    "Touchscreen".Dehner_2;
      S     "Interjack_3";
      A(;
      ON    "Touchscreen".Dehner_3;
      ON    #Inter3_okay;
      );
      R     "Interjack_3";
      A     "Interjack_3";
      =     "Touchscreen".H_Dehner_3;
NETWORK
TITLE = Taster auf der VISU zurücksetzen
      AN    "Jacks_Stop_S";
      R     "Touchscreen".Dehner_3;
NETWORK
TITLE = Wegaufnehmer Dehner 3
      A     "Tur";
      =     L 6.0;
      BLD   103;
      A     "Bipolar";
      =     L 6.1;
      BLD   103;
      CALL  "Scale_mts" (
           PV                       := "Way_Inter3",
           PV_high                  := "Daten DB-2".Inter3Way,
           PV_low                   := 0.000000e+00,
           NB                       := L 6.0,
           Bipolar                  := L 6.1,
           Ueberlauf_High           := "Overflow_High",
           Ueberlauf_Low            := "Overflow_Low",
           Scaled_Value             := "Daten_DB".Inter3_Way);
      NOP   0;
NETWORK
TITLE = Druckaufnehmer Dehner 3
      A     "Tur";
      =     L 6.0;
      BLD   103;
      A     "Bipolar";
      =     L 6.1;
      BLD   103;
      CALL  "Scale_mts" (
           PV                       := "Pres_Inter3",
           PV_high                  := 4.000000e+02,
           PV_low                   := 0.000000e+00,
           NB                       := L 6.0,
           Bipolar                  := L 6.1,
           Ueberlauf_High           := "Overflow_High",
           Ueberlauf_Low            := "Overflow_Low",
           Scaled_Value             := #Druck_Inter3);
      NOP   0;
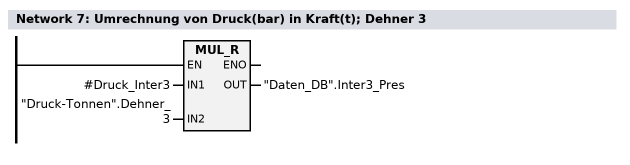
NETWORK
TITLE = Umrechnung von Druck(bar) in Kraft(t); Dehner 3
      L     #Druck_Inter3;
      L     "Druck-Tonnen".Dehner_3;
      *R;
      T     "Daten_DB".Inter3_Pres;
      NOP   0;
END_FUNCTION

FUNCTION "Freigaben" : VOID	// FC 61
TITLE = Freigaben für bestimmte Funktionen
AUTHOR : Simdon
FAMILY : Freigabe
NAME : Release
VERSION : 0.1
BEGIN
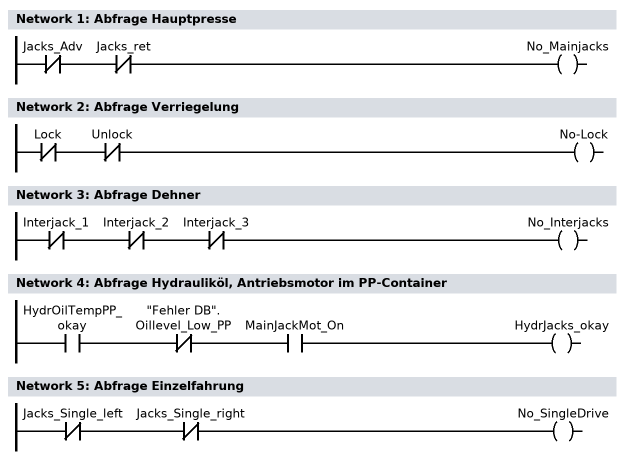
NETWORK
TITLE = Abfrage Hauptpresse
      AN    "Jacks_Adv";
      AN    "Jacks_ret";
      =     "No_Mainjacks";
NETWORK
TITLE = Abfrage Verriegelung
      AN    "Lock";
      AN    "Unlock";
      =     "No-Lock";
NETWORK
TITLE = Abfrage Dehner
      AN    "Interjack_1";
      AN    "Interjack_2";
      AN    "Interjack_3";
      =     "No_Interjacks";
NETWORK
TITLE = Abfrage Hydrauliköl, Antriebsmotor im PP-Container
      A     "HydrOilTempPP_okay";
      AN    "Fehler DB".Oillevel_Low_PP;
      A     "MainJackMot_On";
      =     "HydrJacks_okay";
NETWORK
TITLE = Abfrage Einzelfahrung
      AN    "Jacks_Single_left";
      AN    "Jacks_Single_right";
      =     "No_SingleDrive";
END_FUNCTION

FUNCTION "Betriebsstunden" : VOID	// FC 65
TITLE = Betriebsstundenzähler
AUTHOR : Simdon
FAMILY : System
NAME : BSCount
VERSION : 0.1
VAR_TEMP
  Return_1 : INT ;
  Status_1 : BOOL ;
END_VAR
BEGIN
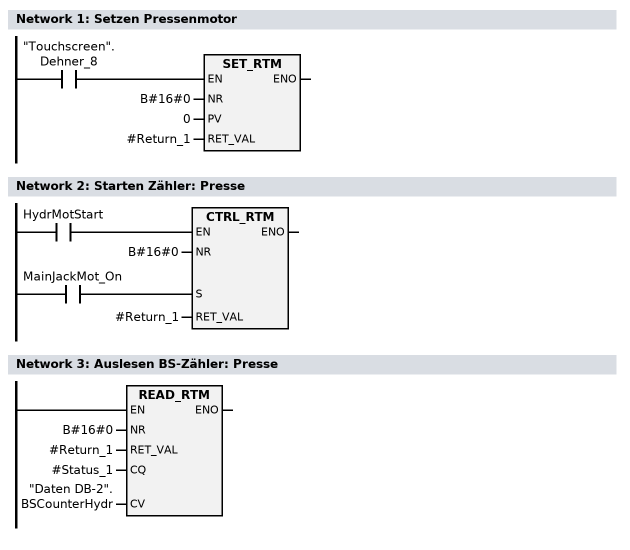
NETWORK
TITLE = Setzen Pressenmotor 
      A     "Touchscreen".Dehner_8;
      JNB   _001;
      CALL  "SET_RTM" (
           NR                       := B#16#0,
           PV                       := 0,
           RET_VAL                  := #Return_1);
_001: NOP   0;
NETWORK
TITLE = Starten Zähler: Presse 
      A     "MainJackMot_On";
      =     L 3.0;
      BLD   103;
      A     "HydrMotStart";
      JNB   _002;
      CALL  "CTRL_RTM" (
           NR                       := B#16#0,
           S                        := L 3.0,
           RET_VAL                  := #Return_1);
_002: NOP   0;
NETWORK
TITLE = Auslesen BS-Zähler: Presse 
      CALL  "READ_RTM" (
           NR                       := B#16#0,
           RET_VAL                  := #Return_1,
           CQ                       := #Status_1,
           CV                       := "Daten DB-2".BSCounterHydr);
      NOP   0;
END_FUNCTION

// FC 68: know-how protected block, not included

FUNCTION "Hydraulik setup" : VOID	// FC 70
AUTHOR : Simdon
FAMILY : Hydr
NAME : Setup
VERSION : 0.1
BEGIN
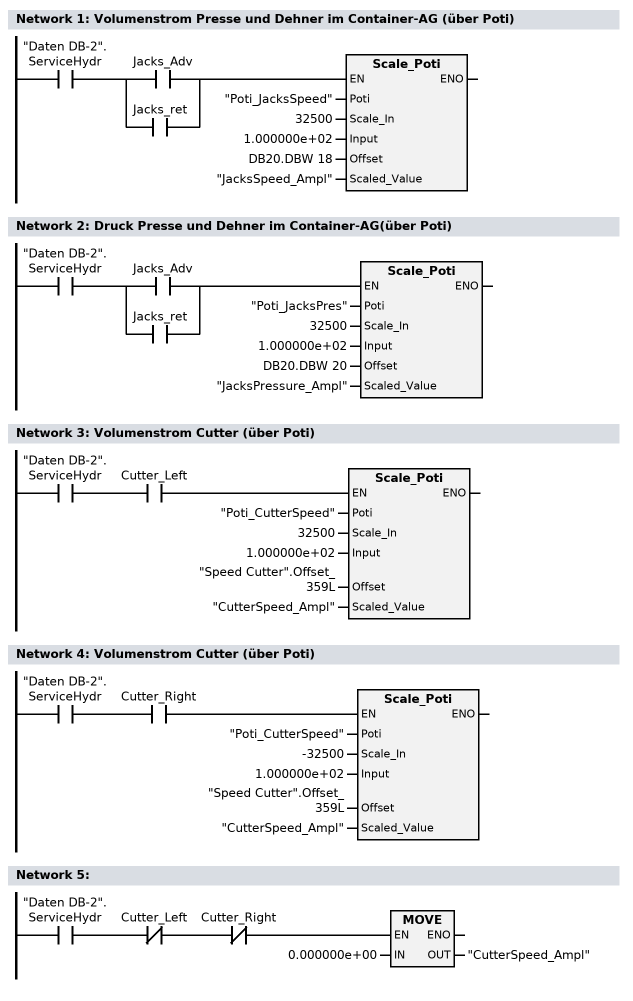
NETWORK
TITLE = Volumenstrom Presse und Dehner im Container-AG (über Poti)
      A     "Daten DB-2".ServiceHydr;
      A(;
      O     "Jacks_Adv";
      O     "Jacks_ret";
      );
      JNB   _001;
      CALL  "Scale_Poti" (
           Poti                     := "Poti_JacksSpeed",
           Scale_In                 := 32500,
           Input                    := 1.000000e+02,
           Offset                   := DB20.DBW 18,
           Scaled_Value             := "JacksSpeed_Ampl");
_001: NOP   0;
NETWORK
TITLE = Druck Presse und Dehner im Container-AG(über Poti)
      A     "Daten DB-2".ServiceHydr;
      A(;
      O     "Jacks_Adv";
      O     "Jacks_ret";
      );
      JNB   _002;
      CALL  "Scale_Poti" (
           Poti                     := "Poti_JacksPres",
           Scale_In                 := 32500,
           Input                    := 1.000000e+02,
           Offset                   := DB20.DBW 20,
           Scaled_Value             := "JacksPressure_Ampl");
_002: NOP   0;
NETWORK
TITLE = Volumenstrom Cutter (über Poti)
      A     "Daten DB-2".ServiceHydr;
      A     "Cutter_Left";
      JNB   _003;
      CALL  "Scale_Poti" (
           Poti                     := "Poti_CutterSpeed",
           Scale_In                 := 32500,
           Input                    := 1.000000e+02,
           Offset                   := "Speed Cutter".Offset_359L,
           Scaled_Value             := "CutterSpeed_Ampl");
_003: NOP   0;
NETWORK
TITLE = Volumenstrom Cutter (über Poti)
      A     "Daten DB-2".ServiceHydr;
      A     "Cutter_Right";
      JNB   _004;
      CALL  "Scale_Poti" (
           Poti                     := "Poti_CutterSpeed",
           Scale_In                 := -32500,
           Input                    := 1.000000e+02,
           Offset                   := "Speed Cutter".Offset_359L,
           Scaled_Value             := "CutterSpeed_Ampl");
_004: NOP   0;
NETWORK
TITLE =
      A     "Daten DB-2".ServiceHydr;
      AN    "Cutter_Left";
      AN    "Cutter_Right";
      JNB   _005;
      L     0.000000e+00;
      T     "CutterSpeed_Ampl";
_005: NOP   0;
END_FUNCTION

FUNCTION "Fehler clr" : VOID	// FC 71
TITLE = Nicht benötigte Fehlermeldungen abschalten
AUTHOR : Simdon
FAMILY : System
NAME : Faults
VERSION : 0.1
BEGIN
NETWORK
TITLE = Fehlermeldungen aus
      CLR;
      =     "Fehler DB".Booster2_Fault;
      =     "Fehler DB".Booster3_Fault;
      =     "Fehler DB".PreMainfilter2_PP;
      =     "Fehler DB".Mainfilter2_PP;
      =     "Fehler DB".LevelSw_Water_BK;
      =     "Fehler DB".HD_Pump;
NETWORK
TITLE = Fehlermeldungen für Bohrkopfaggregat aus
      CLR;
      =     "Fehler DB".CoolPump_EMotor;
      =     "Fehler DB".CoolPump_HydrOil;
      =     "Fehler DB".ThermoCutterMotor;
      =     "Fehler DB".PreReturnlinefilter_BK;
      =     "Fehler DB".PreFedCirFilter_BK;
      =     "Fehler DB".Cool_EMotor_BK;
      =     "Fehler DB".Cool_HydrOil_BK;
      =     "Fehler DB".Oillevel_Med_BK;
      =     "Fehler DB".Oillevel_Low_BK;
      =     "Fehler DB".Returnlinefilter_BK;
      =     "Fehler DB".Warmup_BK;
      =     "Fehler DB".Overheat_BK;
      =     "Fehler DB".Overheat2_BK;
      =     "Fehler DB".FedCirFilter;
      =     "Fehler DB".FedCircuit_BKAG_low;
      =     "Fehler DB".LevelSw_Water_BK;
END_FUNCTION

FUNCTION "Fault3" : VOID	// FC 72
TITLE = Fehlersuche für Pressen- und Schürfradmotor
AUTHOR : Simdon
FAMILY : Faults
NAME : Faults
VERSION : 0.1
BEGIN
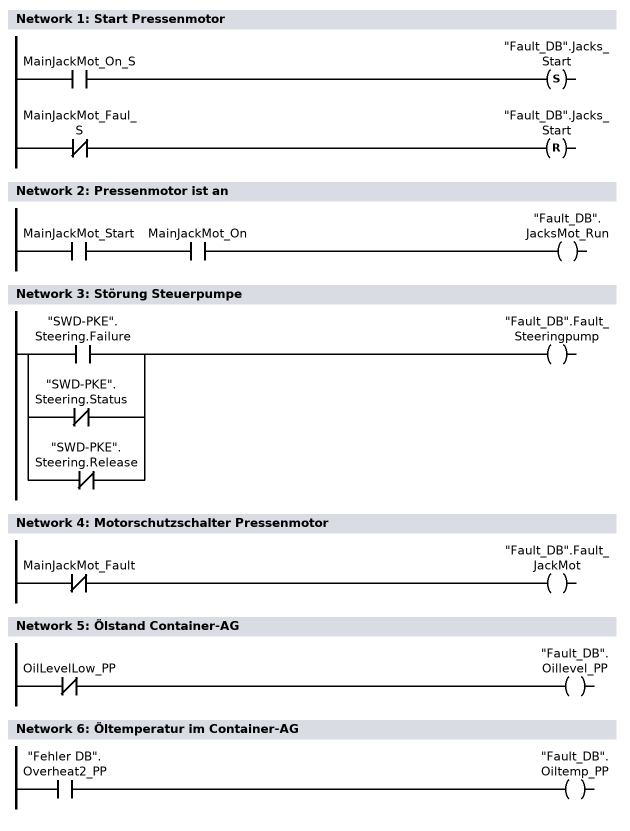
NETWORK
TITLE = Start Pressenmotor
      A     "MainJackMot_On_S";
      S     "Fault_DB".Jacks_Start;
      AN    "MainJackMot_Faul_S";
      R     "Fault_DB".Jacks_Start;
      NOP   0;
NETWORK
TITLE = Pressenmotor ist an
      A     "MainJackMot_Start";
      A     "MainJackMot_On";
      =     "Fault_DB".JacksMot_Run;
NETWORK
TITLE = Störung Steuerpumpe
      O     "SWD-PKE".Steering.Failure;
      ON    "SWD-PKE".Steering.Status;
      ON    "SWD-PKE".Steering.Release;
      =     "Fault_DB".Fault_Steeringpump;
NETWORK
TITLE = Motorschutzschalter Pressenmotor
      AN    "MainJackMot_Fault";
      =     "Fault_DB".Fault_JackMot;
NETWORK
TITLE = Ölstand Container-AG
      AN    "OilLevelLow_PP";
      =     "Fault_DB".Oillevel_PP;
NETWORK
TITLE = Öltemperatur im Container-AG
      A     "Fehler DB".Overheat2_PP;
      =     "Fault_DB".Oiltemp_PP;
END_FUNCTION

FUNCTION "SWD_Pres" : VOID	// FC 73
TITLE = Prüfen ob SWD-Teilnehmer am Bus sind
AUTHOR : Simdon
FAMILY : SWD
NAME : SWD-1
VERSION : 0.1
BEGIN
NETWORK
TITLE = Gruppe 1 der SWD-Teilnehmer
      ON    "S_PowerHead";
      ON    "S_Wing";
      ON    "S_Cylinder_3";
      ON    "S_Cylinder_2";
      ON    "S_Cylinder_1";
      ON    "S_Bypass_open";
      ON    "S_BYpass_close";
      ON    "S_Jet_open";
      =     "SWD_GRP_1";
NETWORK
TITLE =
      ON    "S_Jet_close";
      ON    "S_JacksMot_On";
      ON    "S_JacksMot_Off";
      ON    "S_Charge_On";
      ON    "S_Charge_Off";
      ON    "S_Discharge_Off";
      ON    "S_Discharge_On";
      ON    "S_Booster1_On";
      ON    "S_Booster1_Off";
      ON    "S_Cutter_Mode";
      =     "SWD_GRP_2";
NETWORK
TITLE =
      ON    "S_Jacks_Single";
      ON    "S_Jacks_Mode";
      ON    "S_Locks";
      ON    "S_Jacks_Stop";
      ON    "S_Jacks_Stop";
      ON    "S_Jacks_Advance";
      =     "SWD_GRP_3";
NETWORK
TITLE =
      ON    "S_Cutter_Right";
      ON    "S_Cutter_Stop";
      ON    "S_Cutter_Left";
      =     "SWD_GRP_4";
NETWORK
TITLE = Sammelfehler SWD Gruppe 5
      ON    "DIL_SD";
      ON    "DIL_Head";
      ON    "DIL_OilFan2";
      =     "SWD_GRP_5";
END_FUNCTION

FUNCTION "Protokoll" : VOID	// FC 75
TITLE = Protokollbits
AUTHOR : Simdon
FAMILY : Allg
NAME : Prot
VERSION : 0.1
BEGIN
